# EPICS substitutions: rgamv2/RGA-TS-IOC-01App/Db/RGA-TS-IOC-01.substitutions
#############################################################################
# RGAs
#
# substitutions:
# device  - device name
# port    - serial port (steam device code ie /ty/0/1 => ty_0_1)
# channel - RGA channel number (port number of PC comm port 1-4)
# Controller
#

file rgamv2.template
{
pattern { device       ,   port   }
        { RGA-TS-RGA-01,  ty_41_1 }

}
